// TIA Portal V18 export
FUNCTION_BLOCK "nokButtonMain"   // FB12, FBD
{ S7_Optimized_Access := 'TRUE' }
VERSION : 0.1
// stored: AutoNumber true, IsIECCheckEnabled false, IsRetainMemResEnabled false, MemoryReserve 100, SetENOAutomatically false, UDAEnableTagReadback false
   VAR
      nokButton1 { S7_SetPoint := 'True'} : "nokButton";
      nokButton2 { S7_SetPoint := 'True'} : "nokButton";
      nokButtonQUE_Instance { S7_SetPoint := 'True'} : "nokButtonQUE";
   END_VAR
BEGIN

REGION Network 1: NokButton1
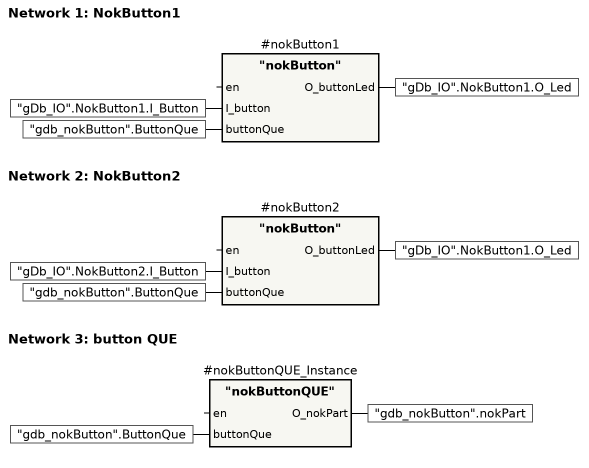
   #nokButton1(I_button := "gDb_IO".NokButton1.I_Button,   // "nokButton"
               buttonQue := "gdb_nokButton".ButtonQue,
               O_buttonLed => "gDb_IO".NokButton1.O_Led);
END_REGION

REGION Network 2: NokButton2
   #nokButton2(I_button := "gDb_IO".NokButton2.I_Button,   // "nokButton"
               buttonQue := "gdb_nokButton".ButtonQue,
               O_buttonLed => "gDb_IO".NokButton1.O_Led);
END_REGION

REGION Network 3: button QUE
   #nokButtonQUE_Instance(buttonQue := "gdb_nokButton".ButtonQue, O_nokPart => "gdb_nokButton".nokPart);   // "nokButtonQUE"
END_REGION
END_FUNCTION_BLOCK
